FUNCTION_BLOCK "fbArchiveEquipShipping"
{ S7_Optimized_Access := 'TRUE' }
VERSION : 0.8
   VAR
      equipmentShipping { ExternalWritable := 'False'} : Array[1..2] of "tEquipment";
   END_VAR

   VAR_TEMP
      tempInt : Int;
   END_VAR


BEGIN
END_FUNCTION_BLOCK

